PROGRAM logcacounters_ex7
VAR
	B11				: DigitalInput_NO;
	B2				: DigitalInput_NO;
	B3				: DigitalInput_NO;
	
	M1				: digitaloutput;
	p1				: digitaloutput;
	P2				: digitaloutput;
	
	teller			: CTUD;
	B1F				: R_trig;
	B2F				: R_trig;
	B3F				: R_trig;
	B2FF			: F_trig;
	
END_VAR

B1F(clk := B11);
B2F(clk := B2);
B3F(clk := B3);
B2FF(clk := B2);


	
//openen en sluiten slagboom
IF B11.isOn THEN
	M1.On();
END_IF
IF B2FF.Q THEN
	M1.Off();
END_IF

END_PROGRAM

(* stored: Version 1.1.0.1
   POU logcacounters_ex7: Id {97827304-5919-4ae7-a0de-0e6999cde2b0}, SpecialFunc None *)
